(* IEC 61131-3 sources: xPLCCore/codesys_code/Application/APP_COMM_FBs, 8 files *)

(* ---- FlyEventActType.st ---- *)
{attribute 'qualified_only'}
{attribute 'strict'}
TYPE FlyEventActType :
(
	NOP := 0,
	PIN_OPERATION := 1,
	PIN_RESET_OPERATION := 2001,

	ACK_SRC_ID := 2002,

	RETURN_ACT := 2342
);
END_TYPE

(* ---- FlyEventData.st ---- *)
TYPE FlyEventData :
STRUCT
	(* Source metadata ------------------------------------------------------ *)
	SourceCommandId : DINT; (* Command that created this fly event. *)

	(* Trigger configuration ------------------------------------------------ *)
	TriggerType : FlyEventTriggerType;

	(* trigger by movement progress ---------------------------------------- *)
	TargetMovementId : SMC_Movement_Id;
	TargetMovementProgress : LREAL;

	(* trigger by distance ------------------------------------------------- *)
	TargetPos_X: LREAL;
	TargetPos_Y: LREAL;
	TargetPos_Z: LREAL;
	TargetDistance: LREAL;
	TriggerInBoundary: BOOL;

	TimeToLiveMs : DINT; (* Optional time (ms) before the trigger auto-expires. -1 = no expiry. *)

	(* Action payload ------------------------------------------------------- *)
	EventId : DINT;
	ActionType : FlyEventActType;

	PinGrp : INT; (* Byte index in the digital output array. *)
	ResetDelayMs : INT; (* Delay (ms) before the reset stage fires. *)
	IoStageCount : INT; (* Number of sequential IO stages configured. *)
	IoStageIndex : INT; (* Next stage index to execute. *)
	IoStageDelayCountdown : DINT; (* Countdown before the next stage fires. *)
	IoStageDelay : ARRAY [0..8] OF DINT; (* Delay (ms) for each stage before it fires. *)
	IoStagePinMask : ARRAY [0..8] OF ULINT; (* Pin mask per stage. *)
	IoStagePinState : ARRAY [0..8] OF ULINT; (* Desired pin state per stage. *)
END_STRUCT
END_TYPE

(* ---- FlyEventTriggerType.st ---- *)
{attribute 'qualified_only'}
{attribute 'strict'}
TYPE FlyEventTriggerType :
(
	NOP := 0,
	MovmentProgressTrigger := 20,
	SequenceDelayWait := 25,

	DistanceTrigger := 120
);
END_TYPE

(* ---- MsgPakInfo.st ---- *)
TYPE MsgPakInfo :
STRUCT
	buf_capacity:UDINT;
	buf_size:UDINT;
	buf:POINTER TO BYTE;

	whead:POINTER TO BYTE;

	useLargeElementCountField:BOOL;
	ele_count:UDINT;

END_STRUCT
END_TYPE

(* ---- Scratchpad_v1.st ---- *)
TYPE Scratchpad_v1 :
STRUCT
    (* Host-owned opaque cursor for crash-and-resume.

       Design contract (decisions_2026-06-22.md §4 (2)):
         - The PLC NEVER interprets any field other than SchemaVersion
           and BootEpoch. Every other field is host-defined opaque
           state. PLC is a durable register, not a brain.
         - schema_version = 0 means "uninitialised / cold-reset wiped".
           PLC writes 1 on first boot. Host treats 0 as invalid and
           goes cold-start.
         - BootEpoch mirrors GVL.BootEpochCount captured at the moment
           of the LAST host write. Host compares on read; mismatch ->
           PLC restarted since the write -> scratchpad is stale ->
           cold-start.

       Memory layout sized to fit comfortably in the SYS reply envelope
       and the retain area budget. Future fields go in `Reserved`. *)
    SchemaVersion     : USINT;
    PlanId            : UDINT;   (* opaque to PLC *)
    PlanIndex         : UDINT;   (* opaque to PLC *)
    IntentKind        : USINT;   (* opaque to PLC -- host-defined enum.
                                    Semantics live in the host (see
                                    `orchestrator/resume.ts` IntentKind);
                                    do NOT branch on this in PLC code,
                                    per memory `plc_stays_generic`. *)
    IntentMovementId  : UDINT;   (* LastAcceptedMovementId at intent write *)
    LastVisionPulse   : UDINT;   (* opaque to PLC *)
    BootEpoch         : UDINT;   (* GVL.BootEpochCount at last write *)
    Reserved          : ARRAY[0..7] OF BYTE;
END_STRUCT
END_TYPE

(* ---- MsgPakInfoClear.st ---- *)
FUNCTION MsgPakInfoClear : BOOL
VAR_IN_OUT
	msgpak:MsgPakInfo;
END_VAR
VAR

END_VAR
(* =========== IMPLEMENTATION =========== *)

msgpak:=MsgPakInfoInit(msgpak.buf,msgpak.buf_capacity,msgpak.useLargeElementCountField);

(* ---- MsgPakInfoInit.st ---- *)
FUNCTION MsgPakInfoInit : MsgPakInfo
VAR_INPUT
	buff:POINTER TO BYTE;
	buffer_size:UDINT;
	useLargeElementCountField:BOOL := TRUE;
END_VAR
VAR

	retStruct:MsgPakInfo;

	mpPacker: FB_MpPacker;
END_VAR
(* =========== IMPLEMENTATION =========== *)

retStruct.buf_capacity:=buffer_size;
retStruct.buf:=buff;
retStruct.useLargeElementCountField:=useLargeElementCountField;
retStruct.ele_count:=0;
retStruct.buf_size:=0;
retStruct.whead := mpPacker.PackMapHeader(pStart := buff, uiCount := TO_UINT(0), bForceLargeField := useLargeElementCountField); // just a place holder
MsgPakInfoInit:=retStruct;

(* ---- MsgPakInfoWrapup.st ---- *)
FUNCTION MsgPakInfoWrapup : BOOL
VAR_IN_OUT
	msgpak:MsgPakInfo;
END_VAR
VAR
	mpPacker: FB_MpPacker;
END_VAR
(* =========== IMPLEMENTATION =========== *)
IF msgpak.useLargeElementCountField=FALSE AND msgpak.ele_count>15 THEN//the size field does not fit
	MsgPakInfoWrapup:=FALSE;
	//TODO: it's possible to move buffer around
	RETURN;
END_IF

mpPacker.PackMapHeader(pStart := msgpak.buf, uiCount := TO_UINT(msgpak.ele_count), bForceLargeField := msgpak.useLargeElementCountField);

MsgPakInfoWrapup:=TRUE;

msgpak.buf_size:=TO_UDINT(msgpak.whead-msgpak.buf);
